FUNCTION_BLOCK ANY2ANY_-715679919 (* Any to any conversion *)
  (* Standard: 61499-2 *)
  (* Version 1.0, 29.10.2008, marumil, nxtControl GmbH, Initial Version *)
  PACKAGE Main;
  (* Compiler Cpp *)
  {SET_ATTRIBUTE(Runtime.FBType.ImplementingType, Runtime.Standard#DYNGEN_ANY2ANY)}
  {SET_ATTRIBUTE(Configuration.GenericFBType.InterfaceParams, Runtime.Standard#CNT:=10;IN${CNT$}:BOOL,BOOL,BOOL,BOOL,BOOL,BOOL,BOOL,BOOL,BOOL,BOOL;OUT${CNT$}:INT,INT,INT,INT,INT,INT,INT,INT,INT,INT)}
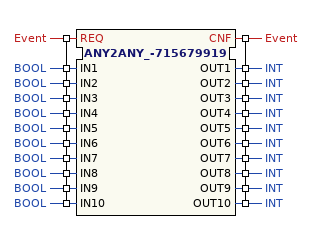
  EVENT_INPUT
    REQ WITH IN1, IN2, IN3, IN4, IN5, IN6, IN7, IN8, IN9, IN10; (* Normal Execution Request *)
  END_EVENT
  EVENT_OUTPUT
    CNF WITH OUT1, OUT2, OUT3, OUT4, OUT5, OUT6, OUT7, OUT8, OUT9, OUT10; (* Execution Confirmation *)
  END_EVENT
  VAR_INPUT
    IN1 : BOOL; (* Argument *)
    IN2 : BOOL; (* Argument *)
    IN3 : BOOL; (* Argument *)
    IN4 : BOOL; (* Argument *)
    IN5 : BOOL; (* Argument *)
    IN6 : BOOL; (* Argument *)
    IN7 : BOOL; (* Argument *)
    IN8 : BOOL; (* Argument *)
    IN9 : BOOL; (* Argument *)
    IN10 : BOOL; (* Argument *)
  END_VAR
  VAR_OUTPUT
    OUT1 : INT; (* Result *)
    OUT2 : INT; (* Result *)
    OUT3 : INT; (* Result *)
    OUT4 : INT; (* Result *)
    OUT5 : INT; (* Result *)
    OUT6 : INT; (* Result *)
    OUT7 : INT; (* Result *)
    OUT8 : INT; (* Result *)
    OUT9 : INT; (* Result *)
    OUT10 : INT; (* Result *)
  END_VAR
  EC_STATES
    START;
  END_STATES
END_FUNCTION_BLOCK
